FUNCTION TryConvert_BYTE_TO_DATE : BOOL
VAR_INPUT
	in : BYTE;
	out : REFERENCE TO DATE;
END_VAR

out := BYTE_TO_DATE(in);
TryConvert_BYTE_TO_DATE := TRUE;

END_FUNCTION

(* stored: Version 1.1.0.1, ProductVersion 3.1.4024.12
   POU TryConvert_BYTE_TO_DATE: Id {d58bf9f8-0b72-4e26-9c64-9c0d052d5d23}, SpecialFunc None *)
